FUNCTION_BLOCK FB_Motor
VAR_INPUT
	mxReset							: BOOL;
	mxEmergency						: BOOL;
	mxAutoMode						: BOOL;
	mxDisableManualAutoTrigger		: BOOL := FALSE; // If this bit is enabled, the outputs status is not changed when change from/to automode happens
END_VAR
VAR_OUTPUT
(*Errors*)
	Errors							: ST_MotorErrors;
	mxErrorInit						: BOOL;		(* Error, stop immediately. Initialisation neccesary *)
	mxErrorStopinPos				: BOOL;		(* Error, stop in position. Only reset neccesary *)

(* State vars *)
	mxCycleBusy						: BOOL;
	mxInitBusy						: BOOL;
	
(* Vars *)
	mxInitialized					: BOOL;
	IsRunning						: BOOL;
	
END_VAR
VAR
	ixThermal						AT %I* : BOOL;
	ixRunning						AT %I* : BOOL;
	ixMaintenance					AT %I* : BOOL;
	Q								AT %Q* : BOOL;
	
	Hmi_On							: BOOL;
	RT_AutoMode						: R_TRIG;
	SR_ErrorThermal					: SR;
	SR_ErrorMaintenance				: SR;
	Ixtest: BOOL;
END_VAR

Error();

(* Reset hmi when switched to automode*)
RT_AutoMode(CLK:= mxAutoMode);

// if manual mode becomes active, the manualmode (hmi) is over written by its current state.
// this ensures that the motor keeps running when it was running and is switched to manual. 
IF RT_AutoMode.Q AND NOT mxDisableManualAutoTrigger THEN Hmi_On:= Q; END_IF	

(* Manual control *)
//IF NOT mxAutoMode THEN Q:= Hmi_On; END_IF

// Is running becomes high when signal becomes low.
IsRunning:= NOT ixRunning;

ACTION Error:
SR_ErrorThermal(SET1:= NOT ixThermal, RESET:= mxReset, Q1=> Errors.Thermal);
SR_ErrorMaintenance(SET1:= NOT ixMaintenance, RESET:= mxReset, Q1=> Errors.Maintenance);

(******************************************************************************************************)
mxErrorStopinPos:= FALSE;
mxErrorInit:= Errors.Thermal OR Errors.Maintenance;
END_ACTION

METHOD M_Init

Q:= FALSE;
END_METHOD

METHOD M_Start : BOOL
VAR_INPUT
END_VAR
Q:=TRUE;

(* Return Value *)
M_Start:= Q;
END_METHOD

METHOD M_Stop : BOOL
VAR_INPUT
END_VAR
Q:= FALSE;

(* Return Value *)
M_Stop:= NOT Q;
END_METHOD

END_FUNCTION_BLOCK

(* stored: Version 1.1.0.1, ProductVersion 3.1.4020.12
   POU FB_Motor: Id {e54d689b-f132-432b-a5ee-ebab27ec5530}, SpecialFunc None
   Action Error: Id {b6eb10cf-ee57-483c-a8e8-0515c9bbf0a7}
   Method M_Init: Id {dcdce6a5-4327-40fe-8dea-aa234b45804b}
   Method M_Start: Id {749247de-8c1d-412c-9de9-805117374cd2}
   Method M_Stop: Id {8ead5074-8d7e-4f90-abd2-910dfc7c8e6c} *)
